// TIA Portal V20 export
FUNCTION_BLOCK "EventsPFE_Recipe"   // FB131, LAD
// stored: MemoryReserve 100, Namespace Unit1.Em8, SetENOAutomatically false
   VAR
      data : Array[1..100] of LReal;
   END_VAR
BEGIN

REGION Network 1: PDR Data41 Recipe - Hipot & Thickness Press Pressure
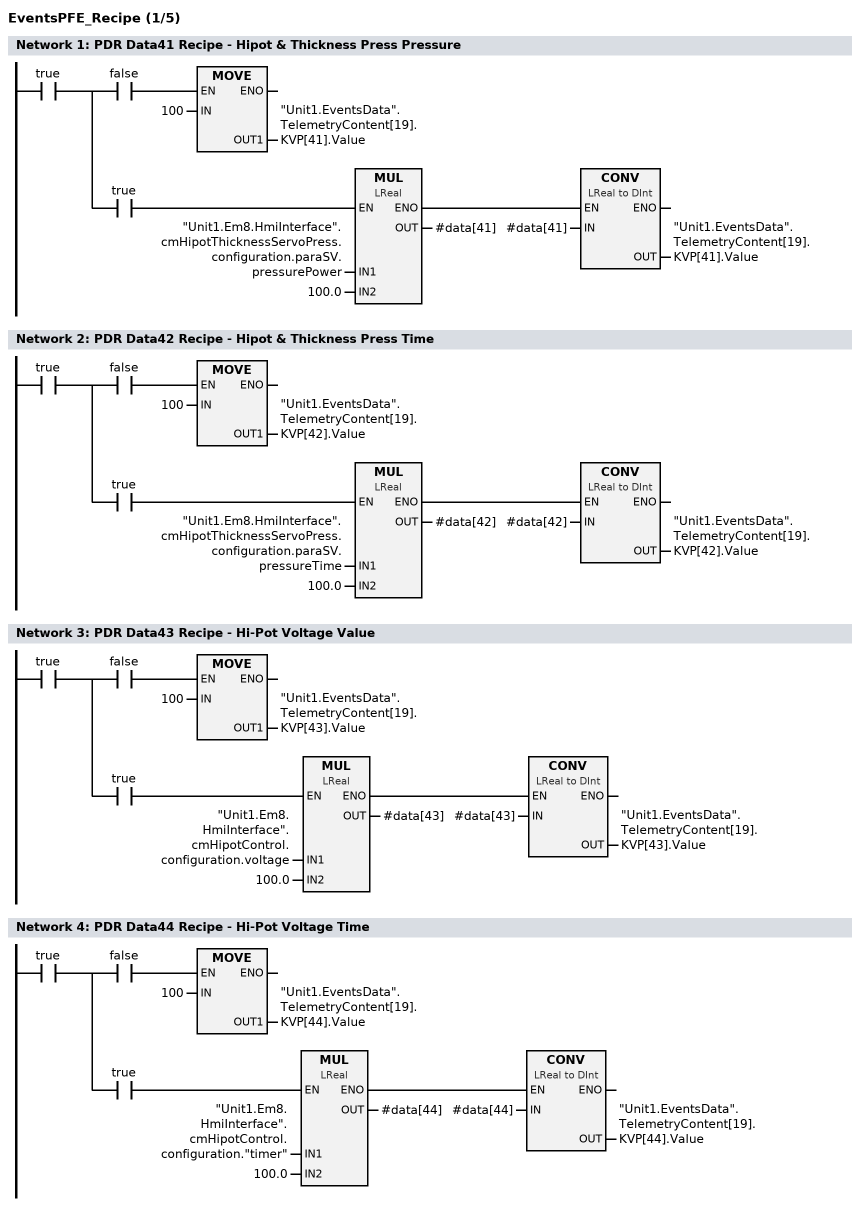
   RUNG wire#powerrail
      Contact( true )
      wire#w1
      Contact( false )
      Move(in := 100, out1 => "Unit1.EventsData".TelemetryContent[19].KVP[41].Value)
   END_RUNG
   RUNG wire#w1
      Contact( true )
      { S7_Templates := "SrcType := LReal" } Mul(in1 := "Unit1.Em8.HmiInterface".cmHipotThicknessServoPress.configuration.paraSV.pressurePower, in2 := 100.0, out => #data[41])
      { S7_Templates := "[SrcType := LReal, DestType := DInt]" } Convert(in := #data[41], out => "Unit1.EventsData".TelemetryContent[19].KVP[41].Value)
   END_RUNG
   // the same network as SCL:
   IF true AND false THEN "Unit1.EventsData".TelemetryContent[19].KVP[41].Value := 100; END_IF;
   IF true AND true THEN
       #data[41] := "Unit1.Em8.HmiInterface".cmHipotThicknessServoPress.configuration.paraSV.pressurePower * 100.0;
       "Unit1.EventsData".TelemetryContent[19].KVP[41].Value := LREAL_TO_DINT(#data[41]);
   END_IF;
END_REGION

REGION Network 2: PDR Data42 Recipe - Hipot & Thickness Press Time
   RUNG wire#powerrail
      Contact( true )
      wire#w1
      Contact( false )
      Move(in := 100, out1 => "Unit1.EventsData".TelemetryContent[19].KVP[42].Value)
   END_RUNG
   RUNG wire#w1
      Contact( true )
      { S7_Templates := "SrcType := LReal" } Mul(in1 := "Unit1.Em8.HmiInterface".cmHipotThicknessServoPress.configuration.paraSV.pressureTime, in2 := 100.0, out => #data[42])
      { S7_Templates := "[SrcType := LReal, DestType := DInt]" } Convert(in := #data[42], out => "Unit1.EventsData".TelemetryContent[19].KVP[42].Value)
   END_RUNG
   // the same network as SCL:
   IF true AND false THEN "Unit1.EventsData".TelemetryContent[19].KVP[42].Value := 100; END_IF;
   IF true AND true THEN
       #data[42] := "Unit1.Em8.HmiInterface".cmHipotThicknessServoPress.configuration.paraSV.pressureTime * 100.0;
       "Unit1.EventsData".TelemetryContent[19].KVP[42].Value := LREAL_TO_DINT(#data[42]);
   END_IF;
END_REGION

REGION Network 3: PDR Data43 Recipe - Hi-Pot Voltage Value
   RUNG wire#powerrail
      Contact( true )
      wire#w1
      Contact( false )
      Move(in := 100, out1 => "Unit1.EventsData".TelemetryContent[19].KVP[43].Value)
   END_RUNG
   RUNG wire#w1
      Contact( true )
      { S7_Templates := "SrcType := LReal" } Mul(in1 := "Unit1.Em8.HmiInterface".cmHipotControl.configuration.voltage, in2 := 100.0, out => #data[43])
      { S7_Templates := "[SrcType := LReal, DestType := DInt]" } Convert(in := #data[43], out => "Unit1.EventsData".TelemetryContent[19].KVP[43].Value)
   END_RUNG
   // the same network as SCL:
   IF true AND false THEN "Unit1.EventsData".TelemetryContent[19].KVP[43].Value := 100; END_IF;
   IF true AND true THEN
       #data[43] := "Unit1.Em8.HmiInterface".cmHipotControl.configuration.voltage * 100.0;
       "Unit1.EventsData".TelemetryContent[19].KVP[43].Value := LREAL_TO_DINT(#data[43]);
   END_IF;
END_REGION

REGION Network 4: PDR Data44 Recipe - Hi-Pot Voltage Time
   RUNG wire#powerrail
      Contact( true )
      wire#w1
      Contact( false )
      Move(in := 100, out1 => "Unit1.EventsData".TelemetryContent[19].KVP[44].Value)
   END_RUNG
   RUNG wire#w1
      Contact( true )
      { S7_Templates := "SrcType := LReal" } Mul(in1 := "Unit1.Em8.HmiInterface".cmHipotControl.configuration."timer", in2 := 100.0, out => #data[44])
      { S7_Templates := "[SrcType := LReal, DestType := DInt]" } Convert(in := #data[44], out => "Unit1.EventsData".TelemetryContent[19].KVP[44].Value)
   END_RUNG
   // the same network as SCL:
   IF true AND false THEN "Unit1.EventsData".TelemetryContent[19].KVP[44].Value := 100; END_IF;
   IF true AND true THEN
       #data[44] := "Unit1.Em8.HmiInterface".cmHipotControl.configuration."timer" * 100.0;
       "Unit1.EventsData".TelemetryContent[19].KVP[44].Value := LREAL_TO_DINT(#data[44]);
   END_IF;
END_REGION

REGION Network 5: PDR Data45 Recipe - Hi-Pot Comp Lower Limit
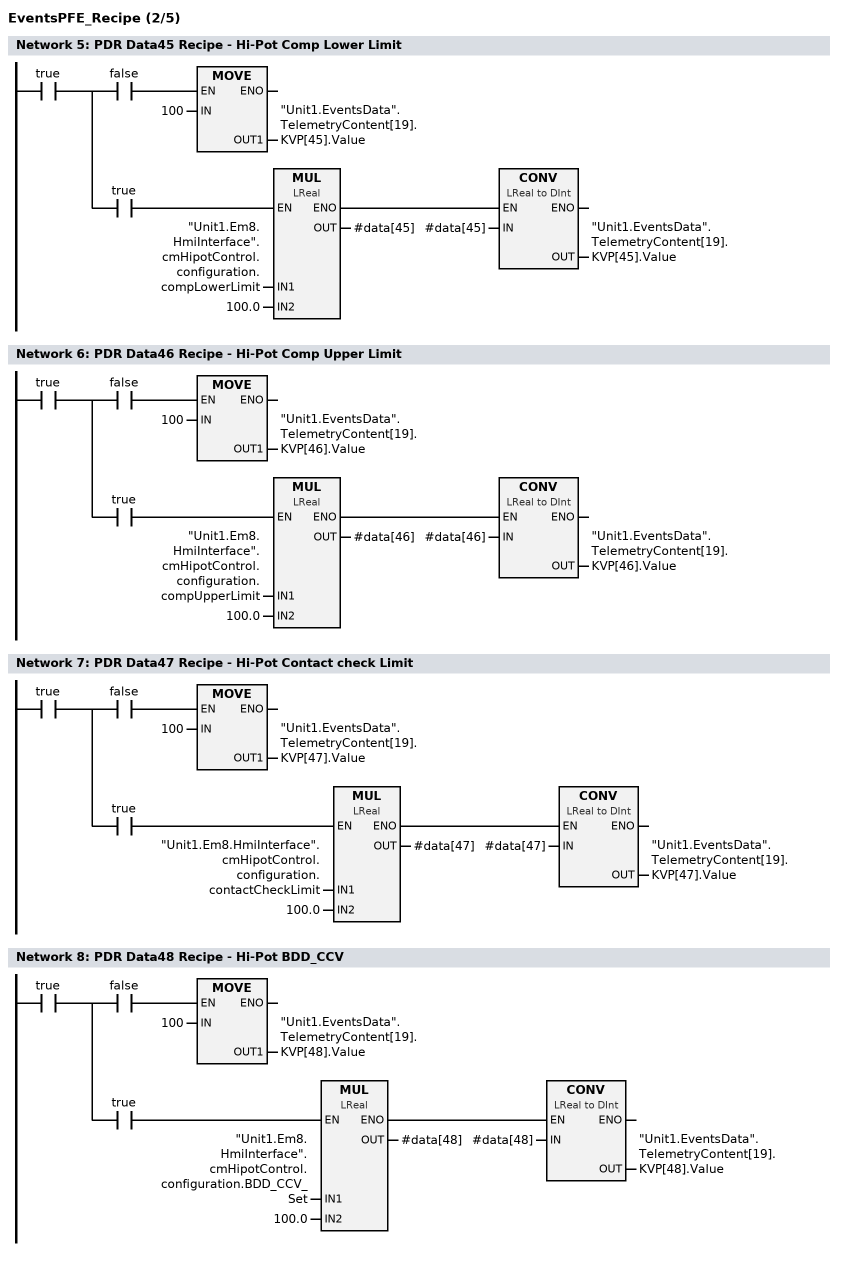
   RUNG wire#powerrail
      Contact( true )
      wire#w1
      Contact( false )
      Move(in := 100, out1 => "Unit1.EventsData".TelemetryContent[19].KVP[45].Value)
   END_RUNG
   RUNG wire#w1
      Contact( true )
      { S7_Templates := "SrcType := LReal" } Mul(in1 := "Unit1.Em8.HmiInterface".cmHipotControl.configuration.compLowerLimit, in2 := 100.0, out => #data[45])
      { S7_Templates := "[SrcType := LReal, DestType := DInt]" } Convert(in := #data[45], out => "Unit1.EventsData".TelemetryContent[19].KVP[45].Value)
   END_RUNG
   // the same network as SCL:
   IF true AND false THEN "Unit1.EventsData".TelemetryContent[19].KVP[45].Value := 100; END_IF;
   IF true AND true THEN
       #data[45] := "Unit1.Em8.HmiInterface".cmHipotControl.configuration.compLowerLimit * 100.0;
       "Unit1.EventsData".TelemetryContent[19].KVP[45].Value := LREAL_TO_DINT(#data[45]);
   END_IF;
END_REGION

REGION Network 6: PDR Data46 Recipe - Hi-Pot Comp Upper Limit
   RUNG wire#powerrail
      Contact( true )
      wire#w1
      Contact( false )
      Move(in := 100, out1 => "Unit1.EventsData".TelemetryContent[19].KVP[46].Value)
   END_RUNG
   RUNG wire#w1
      Contact( true )
      { S7_Templates := "SrcType := LReal" } Mul(in1 := "Unit1.Em8.HmiInterface".cmHipotControl.configuration.compUpperLimit, in2 := 100.0, out => #data[46])
      { S7_Templates := "[SrcType := LReal, DestType := DInt]" } Convert(in := #data[46], out => "Unit1.EventsData".TelemetryContent[19].KVP[46].Value)
   END_RUNG
   // the same network as SCL:
   IF true AND false THEN "Unit1.EventsData".TelemetryContent[19].KVP[46].Value := 100; END_IF;
   IF true AND true THEN
       #data[46] := "Unit1.Em8.HmiInterface".cmHipotControl.configuration.compUpperLimit * 100.0;
       "Unit1.EventsData".TelemetryContent[19].KVP[46].Value := LREAL_TO_DINT(#data[46]);
   END_IF;
END_REGION

REGION Network 7: PDR Data47 Recipe - Hi-Pot Contact check Limit
   RUNG wire#powerrail
      Contact( true )
      wire#w1
      Contact( false )
      Move(in := 100, out1 => "Unit1.EventsData".TelemetryContent[19].KVP[47].Value)
   END_RUNG
   RUNG wire#w1
      Contact( true )
      { S7_Templates := "SrcType := LReal" } Mul(in1 := "Unit1.Em8.HmiInterface".cmHipotControl.configuration.contactCheckLimit, in2 := 100.0, out => #data[47])
      { S7_Templates := "[SrcType := LReal, DestType := DInt]" } Convert(in := #data[47], out => "Unit1.EventsData".TelemetryContent[19].KVP[47].Value)
   END_RUNG
   // the same network as SCL:
   IF true AND false THEN "Unit1.EventsData".TelemetryContent[19].KVP[47].Value := 100; END_IF;
   IF true AND true THEN
       #data[47] := "Unit1.Em8.HmiInterface".cmHipotControl.configuration.contactCheckLimit * 100.0;
       "Unit1.EventsData".TelemetryContent[19].KVP[47].Value := LREAL_TO_DINT(#data[47]);
   END_IF;
END_REGION

REGION Network 8: PDR Data48 Recipe - Hi-Pot BDD_CCV
   RUNG wire#powerrail
      Contact( true )
      wire#w1
      Contact( false )
      Move(in := 100, out1 => "Unit1.EventsData".TelemetryContent[19].KVP[48].Value)
   END_RUNG
   RUNG wire#w1
      Contact( true )
      { S7_Templates := "SrcType := LReal" } Mul(in1 := "Unit1.Em8.HmiInterface".cmHipotControl.configuration.BDD_CCV_Set, in2 := 100.0, out => #data[48])
      { S7_Templates := "[SrcType := LReal, DestType := DInt]" } Convert(in := #data[48], out => "Unit1.EventsData".TelemetryContent[19].KVP[48].Value)
   END_RUNG
   // the same network as SCL:
   IF true AND false THEN "Unit1.EventsData".TelemetryContent[19].KVP[48].Value := 100; END_IF;
   IF true AND true THEN
       #data[48] := "Unit1.Em8.HmiInterface".cmHipotControl.configuration.BDD_CCV_Set * 100.0;
       "Unit1.EventsData".TelemetryContent[19].KVP[48].Value := LREAL_TO_DINT(#data[48]);
   END_IF;
END_REGION

REGION Network 9: PDR Data49 Recipe - Hi-Pot BDD_CVV
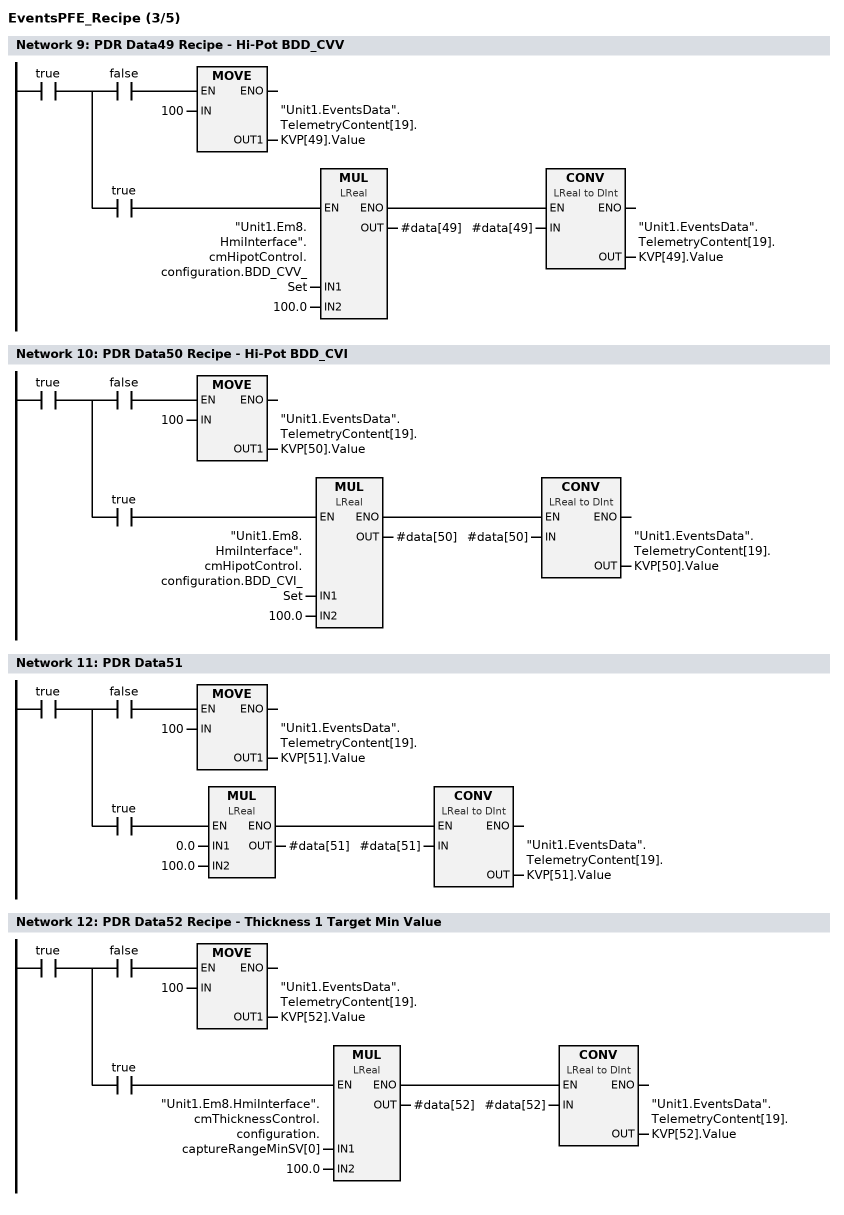
   RUNG wire#powerrail
      Contact( true )
      wire#w1
      Contact( false )
      Move(in := 100, out1 => "Unit1.EventsData".TelemetryContent[19].KVP[49].Value)
   END_RUNG
   RUNG wire#w1
      Contact( true )
      { S7_Templates := "SrcType := LReal" } Mul(in1 := "Unit1.Em8.HmiInterface".cmHipotControl.configuration.BDD_CVV_Set, in2 := 100.0, out => #data[49])
      { S7_Templates := "[SrcType := LReal, DestType := DInt]" } Convert(in := #data[49], out => "Unit1.EventsData".TelemetryContent[19].KVP[49].Value)
   END_RUNG
   // the same network as SCL:
   IF true AND false THEN "Unit1.EventsData".TelemetryContent[19].KVP[49].Value := 100; END_IF;
   IF true AND true THEN
       #data[49] := "Unit1.Em8.HmiInterface".cmHipotControl.configuration.BDD_CVV_Set * 100.0;
       "Unit1.EventsData".TelemetryContent[19].KVP[49].Value := LREAL_TO_DINT(#data[49]);
   END_IF;
END_REGION

REGION Network 10: PDR Data50 Recipe - Hi-Pot BDD_CVI
   RUNG wire#powerrail
      Contact( true )
      wire#w1
      Contact( false )
      Move(in := 100, out1 => "Unit1.EventsData".TelemetryContent[19].KVP[50].Value)
   END_RUNG
   RUNG wire#w1
      Contact( true )
      { S7_Templates := "SrcType := LReal" } Mul(in1 := "Unit1.Em8.HmiInterface".cmHipotControl.configuration.BDD_CVI_Set, in2 := 100.0, out => #data[50])
      { S7_Templates := "[SrcType := LReal, DestType := DInt]" } Convert(in := #data[50], out => "Unit1.EventsData".TelemetryContent[19].KVP[50].Value)
   END_RUNG
   // the same network as SCL:
   IF true AND false THEN "Unit1.EventsData".TelemetryContent[19].KVP[50].Value := 100; END_IF;
   IF true AND true THEN
       #data[50] := "Unit1.Em8.HmiInterface".cmHipotControl.configuration.BDD_CVI_Set * 100.0;
       "Unit1.EventsData".TelemetryContent[19].KVP[50].Value := LREAL_TO_DINT(#data[50]);
   END_IF;
END_REGION

REGION Network 11: PDR Data51
   RUNG wire#powerrail
      Contact( true )
      wire#w1
      Contact( false )
      Move(in := 100, out1 => "Unit1.EventsData".TelemetryContent[19].KVP[51].Value)
   END_RUNG
   RUNG wire#w1
      Contact( true )
      { S7_Templates := "SrcType := LReal" } Mul(in1 := 0.0, in2 := 100.0, out => #data[51])
      { S7_Templates := "[SrcType := LReal, DestType := DInt]" } Convert(in := #data[51], out => "Unit1.EventsData".TelemetryContent[19].KVP[51].Value)
   END_RUNG
   // the same network as SCL:
   IF true AND false THEN "Unit1.EventsData".TelemetryContent[19].KVP[51].Value := 100; END_IF;
   IF true AND true THEN
       #data[51] := 0.0 * 100.0;
       "Unit1.EventsData".TelemetryContent[19].KVP[51].Value := LREAL_TO_DINT(#data[51]);
   END_IF;
END_REGION

REGION Network 12: PDR Data52 Recipe - Thickness 1 Target Min Value
   RUNG wire#powerrail
      Contact( true )
      wire#w1
      Contact( false )
      Move(in := 100, out1 => "Unit1.EventsData".TelemetryContent[19].KVP[52].Value)
   END_RUNG
   RUNG wire#w1
      Contact( true )
      { S7_Templates := "SrcType := LReal" } Mul(in1 := "Unit1.Em8.HmiInterface".cmThicknessControl.configuration.captureRangeMinSV[0], in2 := 100.0, out => #data[52])
      { S7_Templates := "[SrcType := LReal, DestType := DInt]" } Convert(in := #data[52], out => "Unit1.EventsData".TelemetryContent[19].KVP[52].Value)
   END_RUNG
   // the same network as SCL:
   IF true AND false THEN "Unit1.EventsData".TelemetryContent[19].KVP[52].Value := 100; END_IF;
   IF true AND true THEN
       #data[52] := "Unit1.Em8.HmiInterface".cmThicknessControl.configuration.captureRangeMinSV[0] * 100.0;
       "Unit1.EventsData".TelemetryContent[19].KVP[52].Value := LREAL_TO_DINT(#data[52]);
   END_IF;
END_REGION

REGION Network 13: PDR Data53 Recipe - Thickness 2 Target Min Value
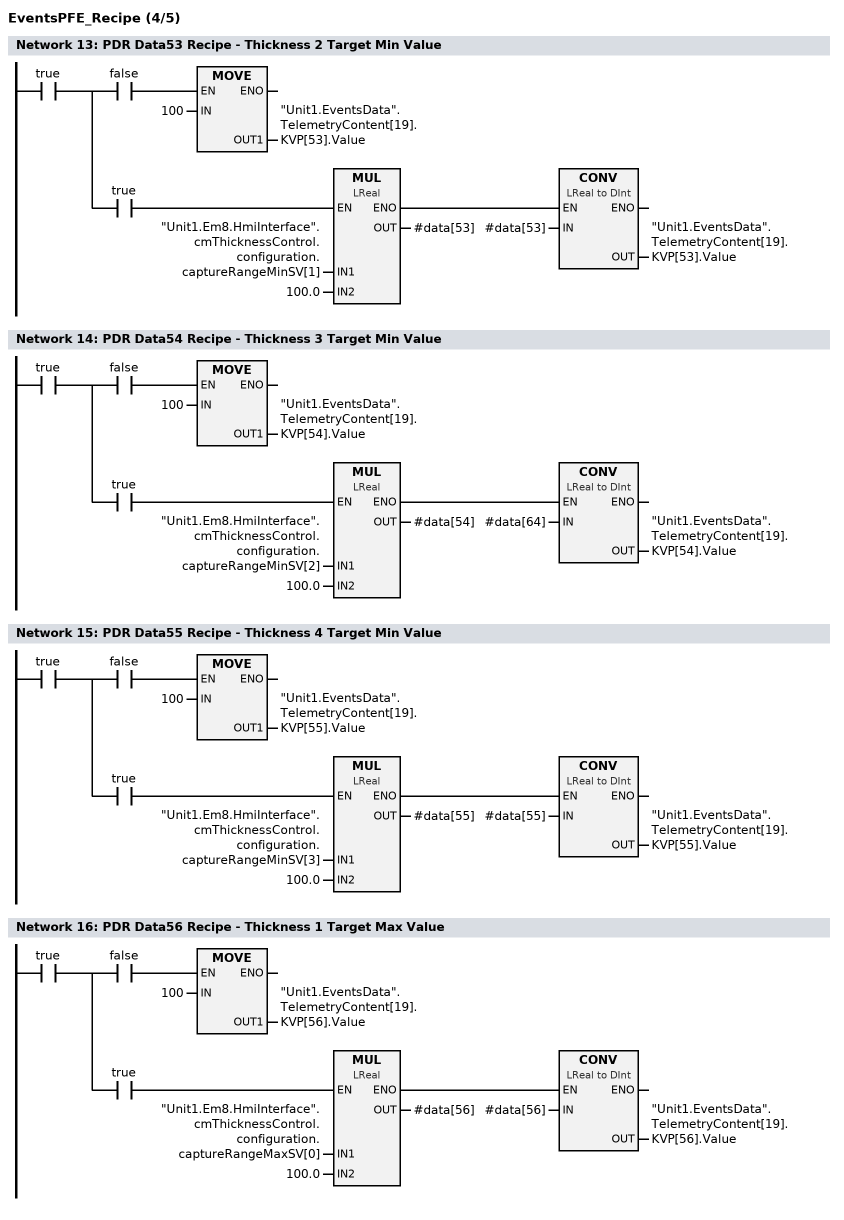
   RUNG wire#powerrail
      Contact( true )
      wire#w1
      Contact( false )
      Move(in := 100, out1 => "Unit1.EventsData".TelemetryContent[19].KVP[53].Value)
   END_RUNG
   RUNG wire#w1
      Contact( true )
      { S7_Templates := "SrcType := LReal" } Mul(in1 := "Unit1.Em8.HmiInterface".cmThicknessControl.configuration.captureRangeMinSV[1], in2 := 100.0, out => #data[53])
      { S7_Templates := "[SrcType := LReal, DestType := DInt]" } Convert(in := #data[53], out => "Unit1.EventsData".TelemetryContent[19].KVP[53].Value)
   END_RUNG
   // the same network as SCL:
   IF true AND false THEN "Unit1.EventsData".TelemetryContent[19].KVP[53].Value := 100; END_IF;
   IF true AND true THEN
       #data[53] := "Unit1.Em8.HmiInterface".cmThicknessControl.configuration.captureRangeMinSV[1] * 100.0;
       "Unit1.EventsData".TelemetryContent[19].KVP[53].Value := LREAL_TO_DINT(#data[53]);
   END_IF;
END_REGION

REGION Network 14: PDR Data54 Recipe - Thickness 3 Target Min Value
   RUNG wire#powerrail
      Contact( true )
      wire#w1
      Contact( false )
      Move(in := 100, out1 => "Unit1.EventsData".TelemetryContent[19].KVP[54].Value)
   END_RUNG
   RUNG wire#w1
      Contact( true )
      { S7_Templates := "SrcType := LReal" } Mul(in1 := "Unit1.Em8.HmiInterface".cmThicknessControl.configuration.captureRangeMinSV[2], in2 := 100.0, out => #data[54])
      { S7_Templates := "[SrcType := LReal, DestType := DInt]" } Convert(in := #data[64], out => "Unit1.EventsData".TelemetryContent[19].KVP[54].Value)
   END_RUNG
   // the same network as SCL:
   IF true AND false THEN "Unit1.EventsData".TelemetryContent[19].KVP[54].Value := 100; END_IF;
   IF true AND true THEN
       #data[54] := "Unit1.Em8.HmiInterface".cmThicknessControl.configuration.captureRangeMinSV[2] * 100.0;
       "Unit1.EventsData".TelemetryContent[19].KVP[54].Value := LREAL_TO_DINT(#data[64]);
   END_IF;
END_REGION

REGION Network 15: PDR Data55 Recipe - Thickness 4 Target Min Value
   RUNG wire#powerrail
      Contact( true )
      wire#w1
      Contact( false )
      Move(in := 100, out1 => "Unit1.EventsData".TelemetryContent[19].KVP[55].Value)
   END_RUNG
   RUNG wire#w1
      Contact( true )
      { S7_Templates := "SrcType := LReal" } Mul(in1 := "Unit1.Em8.HmiInterface".cmThicknessControl.configuration.captureRangeMinSV[3], in2 := 100.0, out => #data[55])
      { S7_Templates := "[SrcType := LReal, DestType := DInt]" } Convert(in := #data[55], out => "Unit1.EventsData".TelemetryContent[19].KVP[55].Value)
   END_RUNG
   // the same network as SCL:
   IF true AND false THEN "Unit1.EventsData".TelemetryContent[19].KVP[55].Value := 100; END_IF;
   IF true AND true THEN
       #data[55] := "Unit1.Em8.HmiInterface".cmThicknessControl.configuration.captureRangeMinSV[3] * 100.0;
       "Unit1.EventsData".TelemetryContent[19].KVP[55].Value := LREAL_TO_DINT(#data[55]);
   END_IF;
END_REGION

REGION Network 16: PDR Data56 Recipe - Thickness 1 Target Max Value
   RUNG wire#powerrail
      Contact( true )
      wire#w1
      Contact( false )
      Move(in := 100, out1 => "Unit1.EventsData".TelemetryContent[19].KVP[56].Value)
   END_RUNG
   RUNG wire#w1
      Contact( true )
      { S7_Templates := "SrcType := LReal" } Mul(in1 := "Unit1.Em8.HmiInterface".cmThicknessControl.configuration.captureRangeMaxSV[0], in2 := 100.0, out => #data[56])
      { S7_Templates := "[SrcType := LReal, DestType := DInt]" } Convert(in := #data[56], out => "Unit1.EventsData".TelemetryContent[19].KVP[56].Value)
   END_RUNG
   // the same network as SCL:
   IF true AND false THEN "Unit1.EventsData".TelemetryContent[19].KVP[56].Value := 100; END_IF;
   IF true AND true THEN
       #data[56] := "Unit1.Em8.HmiInterface".cmThicknessControl.configuration.captureRangeMaxSV[0] * 100.0;
       "Unit1.EventsData".TelemetryContent[19].KVP[56].Value := LREAL_TO_DINT(#data[56]);
   END_IF;
END_REGION

REGION Network 17: PDR Data57 Recipe - Thickness 2 Target Max Value
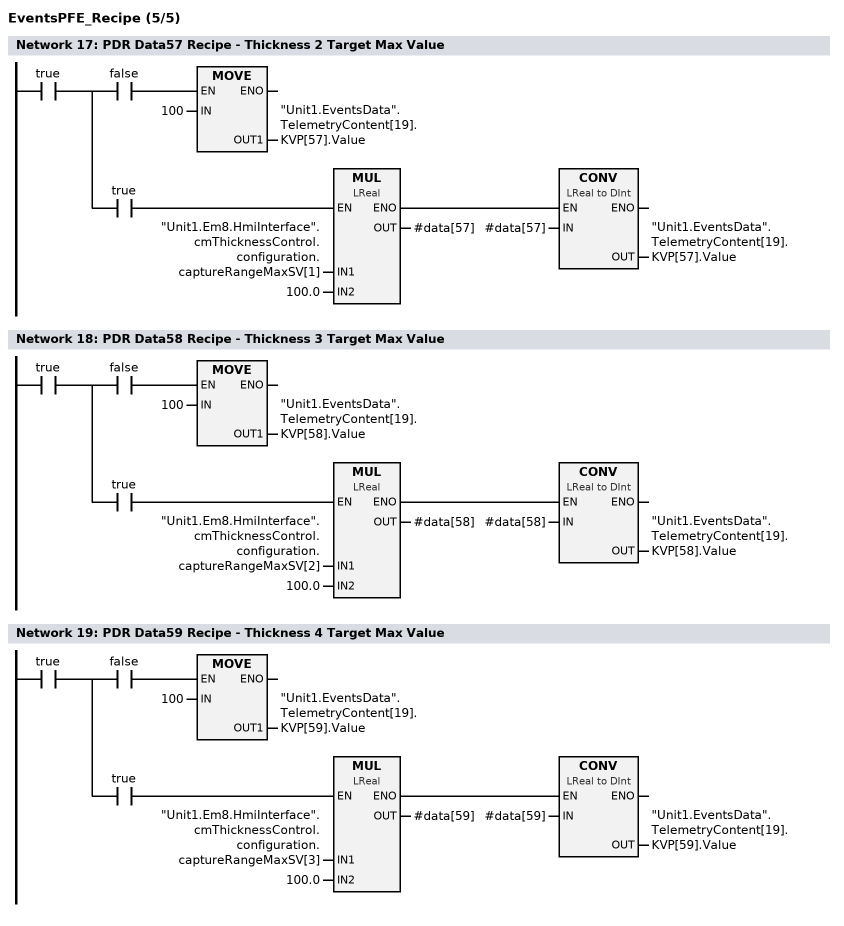
   RUNG wire#powerrail
      Contact( true )
      wire#w1
      Contact( false )
      Move(in := 100, out1 => "Unit1.EventsData".TelemetryContent[19].KVP[57].Value)
   END_RUNG
   RUNG wire#w1
      Contact( true )
      { S7_Templates := "SrcType := LReal" } Mul(in1 := "Unit1.Em8.HmiInterface".cmThicknessControl.configuration.captureRangeMaxSV[1], in2 := 100.0, out => #data[57])
      { S7_Templates := "[SrcType := LReal, DestType := DInt]" } Convert(in := #data[57], out => "Unit1.EventsData".TelemetryContent[19].KVP[57].Value)
   END_RUNG
   // the same network as SCL:
   IF true AND false THEN "Unit1.EventsData".TelemetryContent[19].KVP[57].Value := 100; END_IF;
   IF true AND true THEN
       #data[57] := "Unit1.Em8.HmiInterface".cmThicknessControl.configuration.captureRangeMaxSV[1] * 100.0;
       "Unit1.EventsData".TelemetryContent[19].KVP[57].Value := LREAL_TO_DINT(#data[57]);
   END_IF;
END_REGION

REGION Network 18: PDR Data58 Recipe - Thickness 3 Target Max Value
   RUNG wire#powerrail
      Contact( true )
      wire#w1
      Contact( false )
      Move(in := 100, out1 => "Unit1.EventsData".TelemetryContent[19].KVP[58].Value)
   END_RUNG
   RUNG wire#w1
      Contact( true )
      { S7_Templates := "SrcType := LReal" } Mul(in1 := "Unit1.Em8.HmiInterface".cmThicknessControl.configuration.captureRangeMaxSV[2], in2 := 100.0, out => #data[58])
      { S7_Templates := "[SrcType := LReal, DestType := DInt]" } Convert(in := #data[58], out => "Unit1.EventsData".TelemetryContent[19].KVP[58].Value)
   END_RUNG
   // the same network as SCL:
   IF true AND false THEN "Unit1.EventsData".TelemetryContent[19].KVP[58].Value := 100; END_IF;
   IF true AND true THEN
       #data[58] := "Unit1.Em8.HmiInterface".cmThicknessControl.configuration.captureRangeMaxSV[2] * 100.0;
       "Unit1.EventsData".TelemetryContent[19].KVP[58].Value := LREAL_TO_DINT(#data[58]);
   END_IF;
END_REGION

REGION Network 19: PDR Data59 Recipe - Thickness 4 Target Max Value
   RUNG wire#powerrail
      Contact( true )
      wire#w1
      Contact( false )
      Move(in := 100, out1 => "Unit1.EventsData".TelemetryContent[19].KVP[59].Value)
   END_RUNG
   RUNG wire#w1
      Contact( true )
      { S7_Templates := "SrcType := LReal" } Mul(in1 := "Unit1.Em8.HmiInterface".cmThicknessControl.configuration.captureRangeMaxSV[3], in2 := 100.0, out => #data[59])
      { S7_Templates := "[SrcType := LReal, DestType := DInt]" } Convert(in := #data[59], out => "Unit1.EventsData".TelemetryContent[19].KVP[59].Value)
   END_RUNG
   // the same network as SCL:
   IF true AND false THEN "Unit1.EventsData".TelemetryContent[19].KVP[59].Value := 100; END_IF;
   IF true AND true THEN
       #data[59] := "Unit1.Em8.HmiInterface".cmThicknessControl.configuration.captureRangeMaxSV[3] * 100.0;
       "Unit1.EventsData".TelemetryContent[19].KVP[59].Value := LREAL_TO_DINT(#data[59]);
   END_IF;
END_REGION
END_FUNCTION_BLOCK
